FUNCTION CompareLREAL : BOOL
VAR_INPUT
	Var1	: LREAL;
	Var2	: LREAL;
	Epsilon : LREAL := 1E-6;
END_VAR

CompareLREAL := ABS(Var1 - Var2) < Epsilon;

END_FUNCTION

(* stored: Version 1.1.0.1
   POU CompareLREAL: Id {12f5256c-d8ea-4830-a6bd-8dbd1d000f48}, SpecialFunc None *)
